FUNCTION_BLOCK CylinderDA (* Basic Function Block Type *)
  (* Standard: 61499-2 *)
  (* Version 0.0, 2014-08-21, 4DIAC-IDE, 4DIAC-Consortium *)
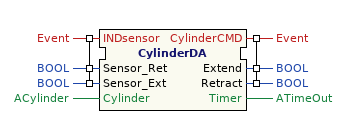
  EVENT_INPUT
    INDsensor WITH Sensor_Ext, Sensor_Ret;
  END_EVENT
  EVENT_OUTPUT
    CylinderCMD WITH Retract, Extend;
  END_EVENT
  VAR_INPUT
    Sensor_Ret : BOOL;
    Sensor_Ext : BOOL;
  END_VAR
  VAR_OUTPUT
    Extend : BOOL;
    Retract : BOOL;
  END_VAR
  SOCKETS
    Cylinder : ACylinder;
  END_SOCKETS
  PLUGS
    Timer : ATimeOut;
  END_PLUGS
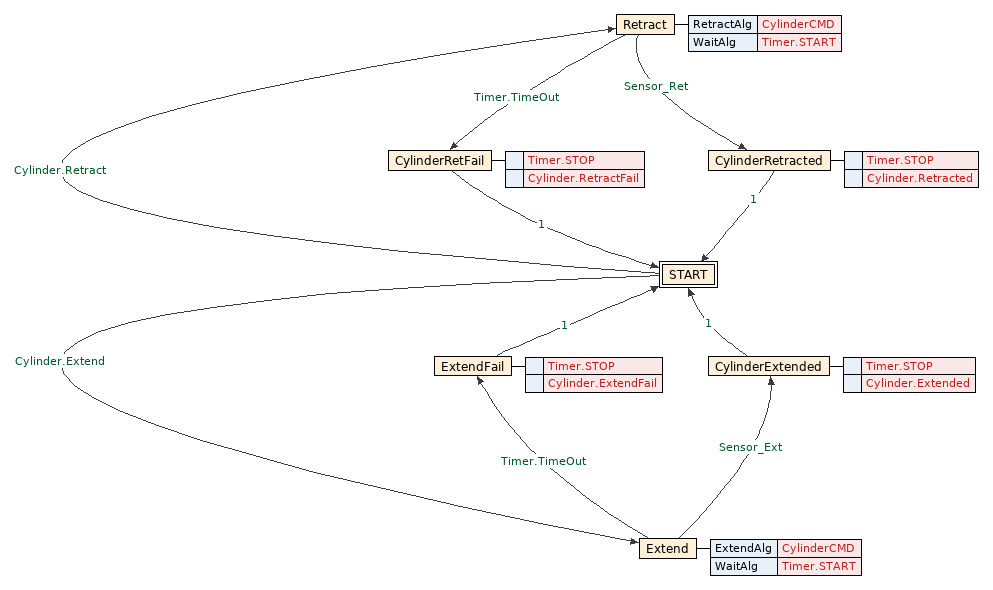
  EC_STATES
    START; (* Initial State *)
    Extend : ExtendAlg -> CylinderCMD, WaitAlg -> Timer.START;
    CylinderExtended : -> Timer.STOP, -> Cylinder.Extended;
    CylinderRetracted : -> Timer.STOP, -> Cylinder.Retracted;
    Retract : RetractAlg -> CylinderCMD, WaitAlg -> Timer.START;
    ExtendFail : -> Timer.STOP, -> Cylinder.ExtendFail;
    CylinderRetFail : -> Timer.STOP, -> Cylinder.RetractFail;
  END_STATES
  EC_TRANSITIONS
    Retract TO CylinderRetFail := Timer.TimeOut;
    Extend TO ExtendFail := Timer.TimeOut;
    Extend TO CylinderExtended := Sensor_Ext;
    Retract TO CylinderRetracted := Sensor_Ret;
    CylinderRetFail TO START := 1;
    CylinderRetracted TO START := 1;
    START TO Retract := Cylinder.Retract;
    CylinderExtended TO START := 1;
    START TO Extend := Cylinder.Extend;
    ExtendFail TO START := 1;
  END_TRANSITIONS
  ALGORITHM RetractAlg IN ST:
Retract := true;
Extend := false;
  END_ALGORITHM
  ALGORITHM ExtendAlg IN ST:
Extend := true;
Retract := false;
  END_ALGORITHM
  ALGORITHM WaitAlg IN ST: (* Timedelay for sensor read *)
Timer.DT := T#5s;
  END_ALGORITHM
END_FUNCTION_BLOCK
